RoboDK station: Celda Robotica.rdk

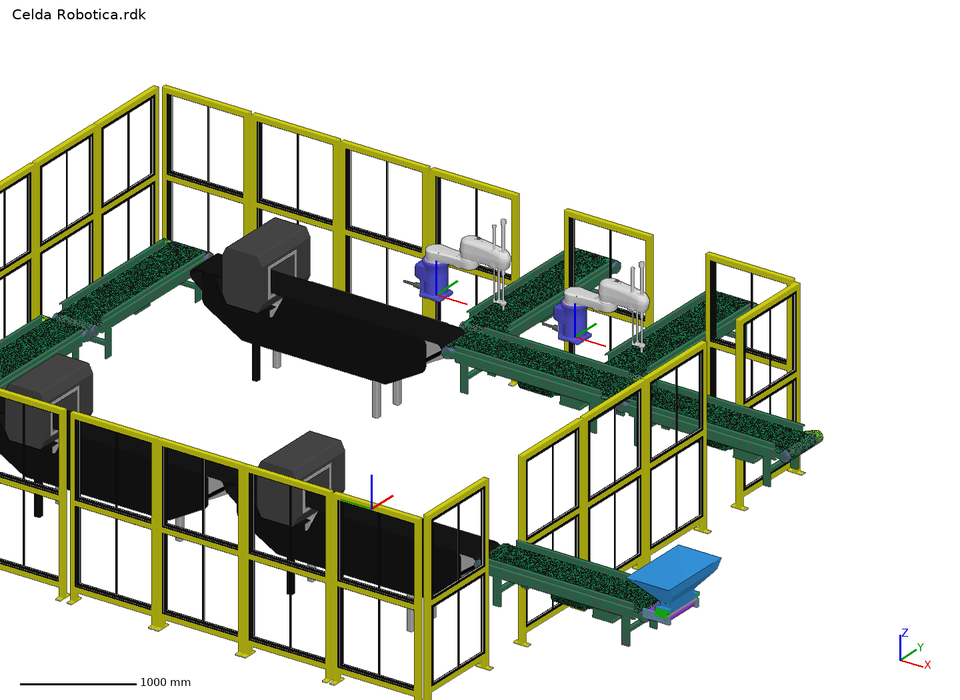
[picture v0: the station drawn from its stored meshes, robots at their saved joint values, targets as dots, program paths as lines]
Station Celda Robotica (saved by RoboDK 5.2.5). Poses are relative to the parent item; angles as X-Y-Z fixed-axis rotations.
  - frame Robot 1 at (-1950, 3750, 0) mm
    - robot Denso HM-4A73: 4 axes, payload 20 kg, reach 700 mm, repeatability 0.022 mm, weight 56 kg
        modified DH rows (alpha deg, a mm, theta deg, d mm): 0, 0, 0, 0; 0, 350, 0, 0; 0, 350, 0, 46 linear; 180, 0, 0, 0
        joint limits [-165, -147, 0, -360] to [165, 147, 300, 360]; home [0, 0, 0, 0]; saved at [0, 0, 0, 0]
  - frame Robot 2 at (-500, 3750, 0) mm
    - robot Denso HM-4A73: 4 axes, payload 20 kg, reach 700 mm, repeatability 0.022 mm, weight 56 kg
        modified DH rows (alpha deg, a mm, theta deg, d mm): 0, 0, 0, 0; 0, 350, 0, 0; 0, 350, 0, 46 linear; 180, 0, 0, 0
        joint limits [-165, -147, 0, -360] to [165, 147, 300, 360]; home [0, 0, 0, 0]; saved at [0, 0, 0, 0]
  - frame Celda Robotica at (0, 0, 0) mm, rotated rx 0 ry 0 rz 90 deg
    - object Tolva_Distribucion_1 at (0, 0, 0) mm, size 480.2 x 432.5 x 787.5 mm, geometry from CONVEYOR WITH HOPPER.STEP
    - object Banda_Suministro_1 at (0, 0, 0) mm, size 527 x 431.8 x 1828.4 mm, geometry from Horizontal belt conveyor.step
    - object Banda_Filtrado_2 at (0, 0, 0) mm, size 2639.7 x 1260 x 880.5 mm, geometry from _ASSY, METAL DETECTOR 1069.STL
    - object Banda_Enjuague_3 at (0, 0, 0) mm, size 2639.7 x 1260 x 880.5 mm, geometry from _ASSY, METAL DETECTOR 1069.STL
    - object Banda_Escurrido_4a at (0, 0, 0) mm, size 527 x 431.8 x 1828.4 mm, geometry from Horizontal belt conveyor.step
    - object Banda_Escurrido_4b at (0, 0, 0) mm, size 527 x 431.8 x 1828.4 mm, geometry from Horizontal belt conveyor.step
    - object Banda_Visio_Artificial_5 at (0, 0, 0) mm, size 2639.7 x 1260 x 880.5 mm, geometry from _ASSY, METAL DETECTOR 1069.STL
    - object Banda_Seleccion_6 at (0, 0, 0) mm, size 527 x 431.8 x 1828.4 mm, geometry from Horizontal belt conveyor.step
    - object Banda_Seleccion_7 at (0, 0, 0) mm, size 527 x 431.8 x 1828.4 mm, geometry from Horizontal belt conveyor.step
    - object Banda_Merma_8a at (0, 0, 0) mm, size 527 x 431.8 x 1828.4 mm, geometry from Horizontal belt conveyor.step
    - object Banda_Merma_8b at (0, 0, 0) mm, size 527 x 431.8 x 1828.4 mm, geometry from Horizontal belt conveyor.step
    - object Barda_Seguridad_9 at (0, 0, 0) mm, size 900 x 1800 x 150 mm, geometry from Security_frame.STEP
      - object BS_9a at (0, 0, 0) mm, size 900 x 1800 x 150 mm, geometry from Security_frame.STEP
      - object BS_9b at (0, 0, 0) mm, size 900 x 1800 x 150 mm, geometry from Security_frame.STEP
      - object BS_9c at (0, 0, 0) mm, size 900 x 1800 x 150 mm, geometry from Security_frame.STEP
      - object BS_9d at (0, 0, 0) mm, size 900 x 1800 x 150 mm, geometry from Security_frame.STEP
      - object BS_9e at (0, 0, 0) mm, size 900 x 1800 x 150 mm, geometry from Security_frame.STEP
      - object BS_9f at (0, 0, 0) mm, size 900 x 1800 x 150 mm, geometry from Security_frame.STEP
      - object BS_9g at (0, 0, 0) mm, size 900 x 1800 x 150 mm, geometry from Security_frame.STEP
      - object BS_9h at (0, 0, 0) mm, size 900 x 1800 x 150 mm, geometry from Security_frame.STEP
      - object BS_9i at (0, 0, 0) mm, size 900 x 1800 x 150 mm, geometry from Security_frame.STEP
      - object BS_9j at (0, 0, 0) mm, size 900 x 1800 x 150 mm, geometry from Security_frame.STEP
      - object BS_9k at (0, 0, 0) mm, size 900 x 1800 x 150 mm, geometry from Security_frame.STEP
      - object BS_9l at (0, 0, 0) mm, size 900 x 1800 x 150 mm, geometry from Security_frame.STEP
      - object BS_9m at (0, 0, 0) mm, size 900 x 1800 x 150 mm, geometry from Security_frame.STEP
      - object BS_9n at (0, 0, 0) mm, size 900 x 1800 x 150 mm, geometry from Security_frame.STEP
      - object BS_9o at (0, 0, 0) mm, size 900 x 1800 x 150 mm, geometry from Security_frame.STEP
      - object BS_9p at (0, 0, 0) mm, size 900 x 1800 x 150 mm, geometry from Security_frame.STEP
      - object BS_9q at (0, 0, 0) mm, size 900 x 1800 x 150 mm, geometry from Security_frame.STEP
      - object BS_9r at (0, 0, 0) mm, size 900 x 1800 x 150 mm, geometry from Security_frame.STEP
      - object BS_9s at (0, 0, 0) mm, size 900 x 1800 x 150 mm, geometry from Security_frame.STEP
      - object BS_9t at (0, 0, 0) mm, size 900 x 1800 x 150 mm, geometry from Security_frame.STEP
      - object BS_9u at (0, 0, 0) mm, size 900 x 1800 x 150 mm, geometry from Security_frame.STEP
      - object BS_9v at (0, 0, 0) mm, size 900 x 1800 x 150 mm, geometry from Security_frame.STEP
      - object BS_9w at (0, 0, 0) mm, size 900 x 1800 x 150 mm, geometry from Security_frame.STEP
